PROGRAM op60_toolchangeover
VAR
	op60_tool_change                    : tool_changeover;
	OP60_TOOL_CHANGE_MODE_SELECTED      : BOOL;
	fb_reset_1                          : BOOL;
	tool_6_fb                           : BOOL;
	tool_8_fb                           : BOOL;
	OP60_TOL_UNLOD_STRT					: BOOL;
	OP60_TOL_LOAD_STRT					: BOOL;
	OP60_TOL_DISENGAGE					: BOOL;
	OP60_TOL_ENGAGE						: BOOL;
	op60_manual_lock                    : BOOL;
	op60_manual_unlock                  : BOOL;
	OP60_UNLD_STUS                      : STRING;
	OP60_LOAD_STUS                      : STRING;
END_VAR

VAR PERSISTENT
	
	OP60_TOL_WRK_POS					: LREAL;
	OP60_TOL_HME_POS					: LREAL;
	op60_TOL_VELOCITY					: LREAL;
	OP60_TOL_CHNGE_CMPLE				: BOOL;
	OP60_TOL_LOAD_COMPLE                : BOOL;
	OP60_TOL_UNLOAD_COMPLE              : BOOL;
	
END_VAR

IF OP60_TOOL_CHANGE_MODE_SELECTED THEN

op60_tool_change(
	actual_pos:=SR60_Vert_servo_ctrl.Actual_Position,
	actual_vel:=SR60_Vert_servo_ctrl.Actual_Velocity,
	target_work_pos:= OP60_TOL_WRK_POS, 
	target_home_pos:= OP60_TOL_HME_POS, 
	target_vel_from_hmi:= op60_TOL_VELOCITY, 
	station_number:= , 
	mover_number:= , 
	no_of_mover_present:= , 
	model_selected:= model_selected, 
	tool_unloading_start:=OP60_TOL_UNLOD_STRT , 
	tool_loading_start:=OP60_TOL_LOAD_STRT , 
	error_active:= , 
	station_in_auto:= OP60_AutoSelected,                   
	station_in_home:=  ,                                   
	absoulte_move_done:= SR60_Vert_servo_ctrl.Axis_In_Pos, 
	tool_6_3_present:= tool_6_fb, 
	tool_7_89_present:= tool_8_fb, 
	fb_reset:=fb_reset_1,
	SERVO_TOL_CHECK_OFFSET_POS := 18, 
	tool_changer_over_complete=> OP60_TOL_CHNGE_CMPLE,
	tool_disengage=> OP60_TOL_DISENGAGE, 
	tool_engagae=> OP60_TOL_ENGAGE, 
	tool_loading_complete=> OP60_TOL_LOAD_COMPLE, 
	tool_unloading_complete=> OP60_TOL_UNLOAD_COMPLE, 
	servo_move_abs=>SR60_Vert_servo_ctrl.ABSmove_Start, 
	unloading_status=>OP60_UNLD_STUS , 
	loading_status=>OP60_LOAD_STUS , 
	target_pos_to_servo=>SR60_Vert_servo_ctrl.Position, 
	target_vel_to_servo=>SR60_Vert_servo_ctrl.Velocity,
    tool_loading_failed := );
	
END_IF	

IF op60_manual_lock OR OP60_TOL_ENGAGE THEN
	O60_TOOL_CHO_UNLOCK_Q1152_2  :=0;
	O60_TOOL_CHO_LOCK_Q1152_3    :=1;
ELSIF op60_manual_unlock OR OP60_TOL_DISENGAGE THEN
	O60_TOOL_CHO_UNLOCK_Q1152_2  :=0;
	O60_TOOL_CHO_LOCK_Q1152_3    :=1;
END_IF

END_PROGRAM

(* stored: Version 1.1.0.1, ProductVersion 3.1.4024.11
   POU op60_toolchangeover: Id {12be9c25-e148-4991-820a-dfe52cad6590}, SpecialFunc None *)
